# EPICS StreamDevice protocol: db/DLCpro.proto
Terminator = LF;
fget = "(param-ref \'laser1:scan:offset)";
fset = "(param-set! \'laser1:scan:offset %f)";

getF{
  out $fget;
  in "%f";
}

setF{
#  @init {in "%f";}
  out $fset;
#  in "%*10c";

}
